{attribute 'linkalways'} 
{attribute 'no_explicit_call' := 'This FB is a CLASS and must be accessed using methods or properties'}
{attribute 'enable_dynamic_creation'}
FUNCTION_BLOCK Node_F_VN_ImageAverageExp EXTENDS VisionNode
VAR
    ipSrcImage : _ITcVnImage;
    aAverage : _TcVnVector4_LREAL;
    ipMask : _ITcVnImage;
    hrPrev : _HRESULT(S_OK);
	hresult : _HRESULT(S_OK);
END_VAR

METHOD PUBLIC  Clone : I_Node
VAR
	pNode : POINTER TO Node_F_VN_ImageAverageExp;
END_VAR
pNode := __NEW(Node_F_VN_ImageAverageExp);
Clone := pNode^;
END_METHOD

METHOD FB_init : BOOL
VAR_INPUT
	bInitRetains : BOOL; // if TRUE, the retain variables are initialized (warm start / cold start)
	bInCopyCode : BOOL;  // if TRUE, the instance afterwards gets moved into the copy code (online change)
END_VAR
AddInput('ipSrcImage', ipSrcImage);
AddInput('ipMask', ipMask);
AddInput('hrPrev', hrPrev);
AddOutput('aAverage', aAverage);
AddOutput('hresult', hresult);
END_METHOD

METHOD PROTECTED OnExecute
hresult.Value := F_VN_ImageAverageExp(
	ipSrcImage := ipSrcImage.Value,
    aAverage := aAverage.Value,
    ipMask := ipMask.Value,
	hrPrev:= hrPrev.Value);
END_METHOD

METHOD PUBLIC PreExecutionCheck
VAR_INPUT
	Check : I_PreExecutionChecks;
END_VAR
Check.IsTrue(ipSrcImage.IsValid, 'ipSrcImage must contain an image');
Check.IsTrue((ipSrcImage.HasChannelCount(1) OR
              ipSrcImage.HasChannelCount(2) OR
              ipSrcImage.HasChannelCount(3) OR
              ipSrcImage.HasChannelCount(4)), 'ipSrcImage must contain 1, 2, 3 or 4 channels');

Check.IsTrue(ipMask.IsValid, 'ipMask must contain an image');
Check.IsTrue(ipMask.HasChannelCount(1), 'ipMask must have 1 channel');
Check.IsTrue(ipMask.IsPixelDepth(8), 'ipMask must have 8 bit pixel depth');
Check.IsTrue(IsImage1SizeEqualToImage2Size(ipMask.Value, ipSrcImage.Value), 'ipMask must be the same size as ipSrcImage');
END_METHOD

END_FUNCTION_BLOCK

(* stored: Version 1.1.0.1, ProductVersion 3.1.4024.13
   POU Node_F_VN_ImageAverageExp: Id {81fc4856-82d3-0881-21ab-b952d9508e80}, SpecialFunc None
   Folder Constructor: Id {0315477e-d9b7-04c1-107e-a84fc6c9ba66}
   Method Clone: Id {294663b8-e998-059c-1d19-2672425b4a99}
   Method FB_init: Id {8ae6bea1-0a66-0cf9-127c-d9e7c66bee14}
   Method OnExecute: Id {5ad77f82-7f1b-0526-3cca-10a8fdcc7321}
   Method PreExecutionCheck: Id {17473ebe-2051-03df-0c28-57b16edca9dd} *)
